{attribute 'GeneratedUsingTerminal: EP1122-0001-0016'}
{attribute addProperty BoxType "EP1122-0001-0016"}
{attribute addProperty Id "A_0025_EP1122_0001_0017A_0025_EP1122_0001_0017_496E3A361450"}
{attribute addProperty CRC "3680443600"}
{attribute addProperty Size "1450"}
TYPE A_0024_EP1122_0001_0016_DB5F1CD0 EXTENDS EP1122_1FC0878B :
STRUCT
	{attribute addProperty Name "A_0025(EP1122-0001-0017)"}
	{attribute addProperty PreviousPort "A_0024(EP1122-0001-0016) : D"}
	A_0025_EP1122_0001_0017 : A_0025_EP1122_0001_0017_496E3A36;
END_STRUCT
END_TYPE

(* stored: Version 1.2.0.0, ProductVersion 3.1.4024.9
   DUT A_0024_EP1122_0001_0016_DB5F1CD0: Id {37c946db-3c27-45e5-9b1a-77b8b6b34e6f} *)
